// TIA Portal V16 export
// export: Created 2021-05-25T16:14:41.0386673Z, ExportSetting WithDefaults, DisplayName Totally Integrated Automation Portal, DisplayVersion V16, DisplayName TIA Portal Version Control Interface, DisplayVersion V16, DisplayName TIA Portal Openness, DisplayVersion V16, DisplayName STEP 7 Professional, DisplayVersion V16, DisplayName STEP 7 Safety, DisplayVersion V16, DisplayName WinCC Unified SCADA Engineering System, DisplayVersion V16
DATA_BLOCK "dbAlarms"   // DB106
{ S7_Optimized_Access := 'FALSE'; DB_Accessible_From_OPC_UA := 'FALSE' }
VERSION : 0.1
// stored: AutoNumber false, DBAccessibleFromOPCUA false, IsOnlyStoredInLoadMemory false, IsWriteProtectedInAS false
   VAR
      PLI : Array[1..4, 1..32] of Bool;
   END_VAR
BEGIN
   PLI[1,1..32] := FALSE;
   PLI[2,1..32] := FALSE;
   PLI[3,1..32] := FALSE;
   PLI[4,1..32] := FALSE;
END_DATA_BLOCK
